// TIA Portal project "scada ile istasyon ürün ayırma factoriy io" (V16)
// Vorlageprojekt für das Buch mit Zielsystem S7-1200

(* hardware
DEVICE "S7-1200-Station_1"  S7-1200 Station
   slot 0: "Baugruppenträger_0"  Rack  V1.0
   slot 1: "PLC_1"  CPU 1214C DC/DC/DC  6ES7 214-1AG40-0XB0  V4.4
   slot 2: "AQ 2x14BIT_1"  SM 1232 AQ2  6ES7 232-4HB32-0XB0  V2.1
DEVICE "PC-System_1"  SIMATIC PC station
   slot 0: "SIMATIC PC station"  Rail  SIMATIC PC-Station  V1.0
      slot 125: "Stationmanager"  Station_Manager  V6.0.4
   slot 1: "HMI_RT_1"  WinCC RT Professional  6AV2 105-0xxxx-xxxx  16.0.0.0
   slot 2: "IE general_1"  IE General  IE_CP  V8.2.0
*)

// ===== PLC "PLC_1"  CPU 1214C DC/DC/DC =====

VAR_GLOBAL   // PLC tag table "ANALOG İNPUTLAR"
   "GÖRÜNTÜ SENSÖRÜ 1" AT %IW30 : Int;
   "GÖRÜNTÜ SENSÖRÜ 2" AT %IW32 : Int;
END_VAR

VAR_GLOBAL   // PLC tag table "OUTPUTLAR"
   "AYIRICI 1" AT %Q0.0 : Bool;
   "AYIRICI 2" AT %Q0.1 : Bool;
   "KONVEYÖR  1" AT %Q0.2 : Bool;
   "KONVEYÖR  2" AT %Q0.3 : Bool;
   "KONVEYÖR  3" AT %Q0.4 : Bool;
   "KONVEYÖR  4" AT %Q0.5 : Bool;
END_VAR

VAR_GLOBAL   // PLC tag table "İNPUTLAR"
   "SENSÖR 1" AT %I0.0 : Bool;
   "SENSÖR 2" AT %I0.1 : Bool;
   "SENSÖR 3" AT %I0.2 : Bool;
   "SENSÖR 4" AT %I0.3 : Bool;
   "AYIRICI 1 GERİ SENSÖRÜ" AT %I0.4 : Bool;
   "AYIRICI 1 İLERİ SENSÖRÜ" AT %I0.5 : Bool;
   "AYIRICI 2 GERİ SENSÖRÜ" AT %I0.6 : Bool;
   "AYIRICI 2 İLERİ SENSÖRÜ" AT %I0.7 : Bool;
END_VAR

DATA_BLOCK "DATALAR"   // DB1
{ S7_Optimized_Access := 'TRUE' }
VERSION : 0.1
   VAR
      "SİSTEM START" : Bool;
      "SİSTEM STOP" : Bool;
      "SİSTEM RESET" : Bool;
      "SİSTEM GENEL MEM" : Bool;
      "YESİL ÜRÜN SAYISI" : Int;
      "MAVİ ÜRÜN SAYISI" : Int;
      "TOPLAM ÜRÜN SAYISI" : Int;
      "AYRILACAK ÜRÜN SAYISI" : Int;
      M1 : Bool;
      M2 : Bool;
      M3 : Bool;
      M4 : Bool;
      "AYRICI DURUM BİL MEM" : Bool;
      "M3_GRT 1 MAVİ" : Bool;
      "M3_GRT 1 YESİL" : Bool;
      "M3_GRT  2 MAVİ" : Bool;
      "M3_GRT 2  YESİL" : Bool;
      TEMP_1 : Bool;
      TEMP_2 : Bool;
      TEMP_3 : Bool;
      TEMP_4 : Bool;
      TEMP_5 : Bool;
      TEMP_6 : Bool;
      TEMP_7 : Bool;
      TEMP_8 : Bool;
      TEMP_9 : Bool;
   END_VAR
BEGIN
END_DATA_BLOCK

// folder: System blocks/Program resources

DATA_BLOCK "TİME 1"   // DB2
{ S7_Optimized_Access := 'TRUE' }
AUTHOR : Simatic
FAMILY : IEC
NAME : IEC_TMR
VERSION : 1.0
// stored: InstanceOfName IEC_TIMER
"IEC_TIMER"
BEGIN
END_DATA_BLOCK

DATA_BLOCK "TİME 2"   // DB3
{ S7_Optimized_Access := 'TRUE' }
AUTHOR : Simatic
FAMILY : IEC
NAME : IEC_TMR
VERSION : 1.0
// stored: InstanceOfName IEC_TIMER
"IEC_TIMER"
BEGIN
END_DATA_BLOCK

DATA_BLOCK "tİME 3"   // DB4
{ S7_Optimized_Access := 'TRUE' }
AUTHOR : Simatic
FAMILY : IEC
NAME : IEC_TMR
VERSION : 1.0
// stored: InstanceOfName IEC_TIMER
"IEC_TIMER"
BEGIN
END_DATA_BLOCK

DATA_BLOCK "SAYICI 1"   // DB5
{ S7_Optimized_Access := 'TRUE' }
AUTHOR : Simatic
FAMILY : IEC
NAME : CNTR
VERSION : 1.0
// stored: InstanceOfName IEC_COUNTER
"IEC_COUNTER"
BEGIN
END_DATA_BLOCK

// folder: (top level)

FUNCTION "MHJ-PLC-Lab-Function-S71200" : Void   // FC9000, SCL
{ S7_Optimized_Access := 'TRUE' }
VERSION : 0.1
   VAR_TEMP
      rdTimeReturn : Int;
      outputTime : DTL;
      SyncVal : Byte;
      forVal : Int;
      forVal_2 : Int;
      Value : Byte;
   END_VAR
   VAR CONSTANT
      CompVal : Byte := 16#34;
      Value_01 : Byte := 16#11;
      Value_01_DW : DWord := 16#A165_D992;
      Value_02_DW : DWord := 16#58BE_4401;
   END_VAR
BEGIN

   #Value:=PEEK(area := 16#82,
        dbNumber := 0,
        byteOffset := 511);
   #Value := #Value + 1;

   POKE(area := 16#82,
        dbNumber := 0,
        byteOffset := 511,
        value := #Value);

   POKE(area:=16#81,
        dbNumber:=0,
        byteOffset:=1016,
        value:=#Value_01_DW);
   POKE(area := 16#81,
        dbNumber := 0,
        byteOffset := 1020,
        value := #Value_02_DW);

   POKE(area := 16#81,
        dbNumber := 0,
        byteOffset := 511,
        value := B#16#00);

   FOR #forVal := 0 TO 120 DO
       FOR #forVal_2:=0 TO 10 DO
           #rdTimeReturn:=RD_SYS_T(#outputTime);
           #rdTimeReturn := WR_SYS_T(#outputTime);
           #rdTimeReturn := RD_SYS_T(#outputTime);
           #rdTimeReturn := WR_SYS_T(#outputTime);
       END_FOR;
       #SyncVal:= PEEK(area := 16#81,
                      dbNumber := 0,
                      byteOffset := 511);
       IF #SyncVal = #CompVal THEN
          GOTO M_1;
       END_IF;
   END_FOR;
   RETURN;

   M_1:
   POKE(area := 16#81,
        dbNumber := 0,
        byteOffset := 511,
        value := B#16#0);
END_FUNCTION

ORGANIZATION_BLOCK "Main"   // OB1, LAD, ProgramCycle
TITLE = "Main Program Sweep (Cycle)"
{ S7_Optimized_Access := 'TRUE' }
VERSION : 0.1
   VAR_INPUT
      Initial_Call : Bool;   // Initial call of this OB
      Remanence : Bool;   // =True, if remanent data are available
   END_VAR
   VAR_TEMP   // added for the SCL form of the ladder/FBD networks
      _w1 : Bool;
      _w2 : Bool;
      _w3 : Bool;
   END_VAR
BEGIN

REGION Network 1: Konnektierungsbaustein für PLC-Lab
   // Im Netzwerk 1 wird der Konnektierungsbaustein für PLC-Lab aufgerufen.
   // Dieser Aufruf darf nicht entfernt werden!
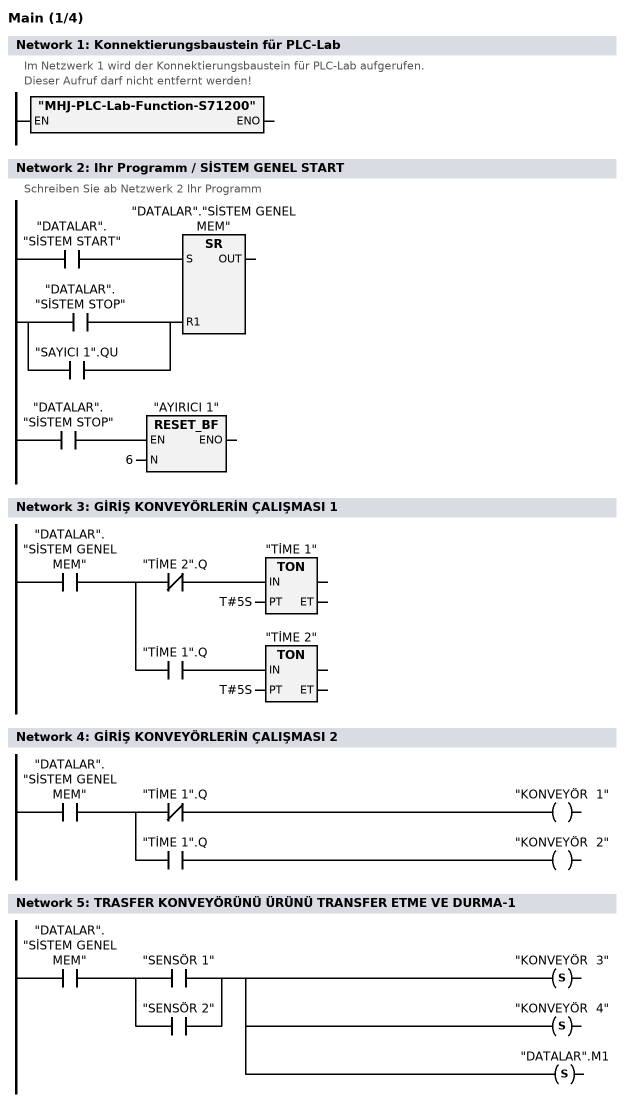
   RUNG wire#powerrail
      "MHJ-PLC-Lab-Function-S71200"()
   END_RUNG
   // the same network as SCL:
   "MHJ-PLC-Lab-Function-S71200"();
END_REGION

REGION Network 2: Ihr Programm / SİSTEM GENEL START
   // Schreiben Sie ab Netzwerk 2 Ihr Programm
   // no SCL statement known for RBitfield: written as a call
   IF "DATALAR"."SİSTEM START" THEN
       "DATALAR"."SİSTEM GENEL MEM" := TRUE;   // SR flip-flop
   END_IF;
   IF "DATALAR"."SİSTEM STOP" OR "SAYICI 1".QU THEN "DATALAR"."SİSTEM GENEL MEM" := FALSE; END_IF;
   IF "DATALAR"."SİSTEM STOP" THEN RESET_BF(operand := "AYIRICI 1", n := 6); END_IF;
END_REGION

REGION Network 3: GİRİŞ KONVEYÖRLERİN ÇALIŞMASI 1
   "TİME 1".TON(IN := "DATALAR"."SİSTEM GENEL MEM" AND NOT "TİME 2".Q, PT := T#5S);
   "TİME 2".TON(IN := "DATALAR"."SİSTEM GENEL MEM" AND "TİME 1".Q, PT := T#5S);
END_REGION

REGION Network 4: GİRİŞ KONVEYÖRLERİN ÇALIŞMASI 2
   RUNG wire#powerrail
      Contact( "DATALAR"."SİSTEM GENEL MEM" )
      wire#w1
      I_Contact( "TİME 1".Q )
      Coil( "KONVEYÖR  1" )
   END_RUNG
   RUNG wire#w1
      Contact( "TİME 1".Q )
      Coil( "KONVEYÖR  2" )
   END_RUNG
   // the same network as SCL:
   "KONVEYÖR  1" := "DATALAR"."SİSTEM GENEL MEM" AND NOT "TİME 1".Q;
   "KONVEYÖR  2" := "DATALAR"."SİSTEM GENEL MEM" AND "TİME 1".Q;
END_REGION

REGION Network 5: TRASFER KONVEYÖRÜNÜ ÜRÜNÜ TRANSFER ETME VE DURMA-1
   RUNG wire#powerrail
      Contact( "DATALAR"."SİSTEM GENEL MEM" )
      wire#w1
      Contact( "SENSÖR 1" )
      wire#w2
      S_Coil( "KONVEYÖR  3" )
   END_RUNG
   RUNG wire#w1
      Contact( "SENSÖR 2" )
   END_RUNG wire#w2
   RUNG wire#w2
      S_Coil( "KONVEYÖR  4" )
   END_RUNG
   RUNG wire#w2
      S_Coil( "DATALAR".M1 )
   END_RUNG
   // the same network as SCL:
   IF "DATALAR"."SİSTEM GENEL MEM" AND ("SENSÖR 1" OR "SENSÖR 2") THEN
       "KONVEYÖR  3" := TRUE;
       "KONVEYÖR  4" := TRUE;
       "DATALAR".M1 := TRUE;
   END_IF;
END_REGION

REGION Network 6: TRASFER KONVEYÖRÜNÜ ÜRÜNÜ TRANSFER ETME VE DURMA-2
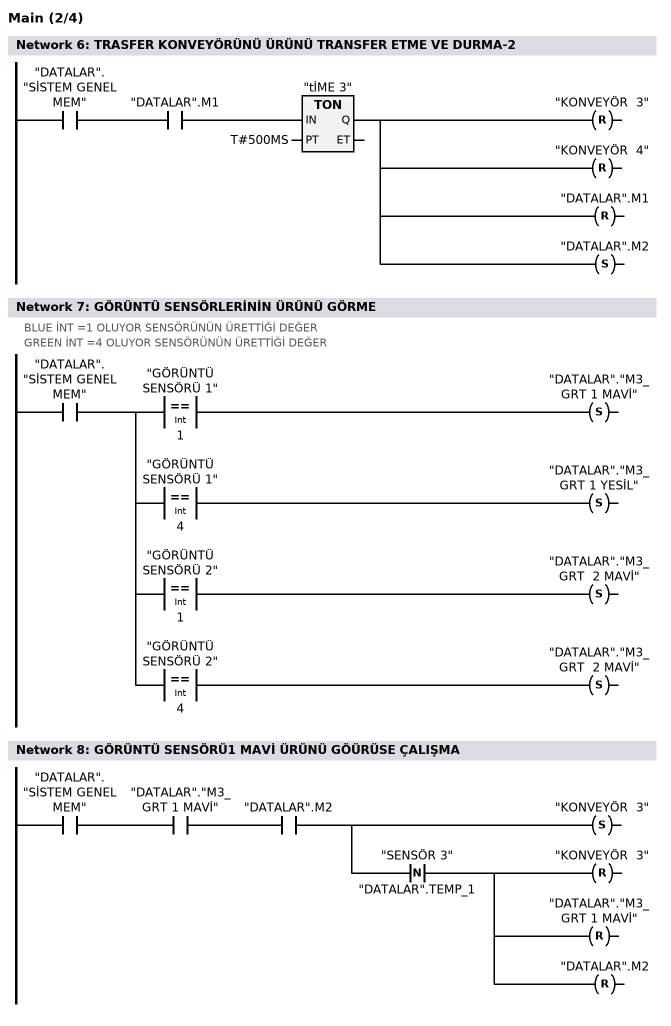
   "tİME 3".TON(IN := "DATALAR"."SİSTEM GENEL MEM" AND "DATALAR".M1, PT := T#500MS);
   IF "tİME 3".Q THEN
       "KONVEYÖR  3" := FALSE;
       "KONVEYÖR  4" := FALSE;
       "DATALAR".M1 := FALSE;
       "DATALAR".M2 := TRUE;
   END_IF;
END_REGION

REGION Network 7: GÖRÜNTÜ SENSÖRLERİNİN ÜRÜNÜ GÖRME
   // BLUE İNT =1 OLUYOR SENSÖRÜNÜN ÜRETTİĞİ DEĞER
   // GREEN İNT =4 OLUYOR SENSÖRÜNÜN ÜRETTİĞİ DEĞER
   RUNG wire#powerrail
      Contact( "DATALAR"."SİSTEM GENEL MEM" )
      wire#w1
      { S7_Templates := "SrcType := Int" } EQ_Contact(in1 := "GÖRÜNTÜ SENSÖRÜ 1", in2 := 1)
      S_Coil( "DATALAR"."M3_GRT 1 MAVİ" )
   END_RUNG
   RUNG wire#w1
      { S7_Templates := "SrcType := Int" } EQ_Contact(in1 := "GÖRÜNTÜ SENSÖRÜ 1", in2 := 4)
      S_Coil( "DATALAR"."M3_GRT 1 YESİL" )
   END_RUNG
   RUNG wire#w1
      { S7_Templates := "SrcType := Int" } EQ_Contact(in1 := "GÖRÜNTÜ SENSÖRÜ 2", in2 := 1)
      S_Coil( "DATALAR"."M3_GRT  2 MAVİ" )
   END_RUNG
   RUNG wire#w1
      { S7_Templates := "SrcType := Int" } EQ_Contact(in1 := "GÖRÜNTÜ SENSÖRÜ 2", in2 := 4)
      S_Coil( "DATALAR"."M3_GRT  2 MAVİ" )
   END_RUNG
   // the same network as SCL:
   IF "DATALAR"."SİSTEM GENEL MEM" AND ("GÖRÜNTÜ SENSÖRÜ 1" = 1) THEN
       "DATALAR"."M3_GRT 1 MAVİ" := TRUE;
   END_IF;
   IF "DATALAR"."SİSTEM GENEL MEM" AND ("GÖRÜNTÜ SENSÖRÜ 1" = 4) THEN
       "DATALAR"."M3_GRT 1 YESİL" := TRUE;
   END_IF;
   IF "DATALAR"."SİSTEM GENEL MEM" AND ("GÖRÜNTÜ SENSÖRÜ 2" = 1) THEN
       "DATALAR"."M3_GRT  2 MAVİ" := TRUE;
   END_IF;
   IF "DATALAR"."SİSTEM GENEL MEM" AND ("GÖRÜNTÜ SENSÖRÜ 2" = 4) THEN
       "DATALAR"."M3_GRT  2 MAVİ" := TRUE;
   END_IF;
END_REGION

REGION Network 8: GÖRÜNTÜ SENSÖRÜ1 MAVİ ÜRÜNÜ GÖÜRÜSE ÇALIŞMA
   RUNG wire#powerrail
      Contact( "DATALAR"."SİSTEM GENEL MEM" )
      Contact( "DATALAR"."M3_GRT 1 MAVİ" )
      Contact( "DATALAR".M2 )
      wire#w1
      S_Coil( "KONVEYÖR  3" )
   END_RUNG
   RUNG wire#w1
      N_Contact(operand := "SENSÖR 3", bit := "DATALAR".TEMP_1)
      wire#w2
      R_Coil( "KONVEYÖR  3" )
   END_RUNG
   RUNG wire#w2
      R_Coil( "DATALAR"."M3_GRT 1 MAVİ" )
   END_RUNG
   RUNG wire#w2
      R_Coil( "DATALAR".M2 )
   END_RUNG
   // the same network as SCL:
   #_w1 := "DATALAR"."SİSTEM GENEL MEM" AND "DATALAR"."M3_GRT 1 MAVİ" AND "DATALAR".M2;
   IF #_w1 THEN "KONVEYÖR  3" := TRUE; END_IF;
   #_w2 := #_w1 AND NOT "SENSÖR 3" AND "DATALAR".TEMP_1;   // falling edge of "SENSÖR 3"
   "DATALAR".TEMP_1 := "SENSÖR 3";
   IF #_w2 THEN
       "KONVEYÖR  3" := FALSE;
       "DATALAR"."M3_GRT 1 MAVİ" := FALSE;
       "DATALAR".M2 := FALSE;
   END_IF;
END_REGION

REGION Network 9: GÖRÜNTÜ SENSÖRÜ1 YEŞİL ÜRÜNÜ GÖÜRÜSE ÇALIŞMA
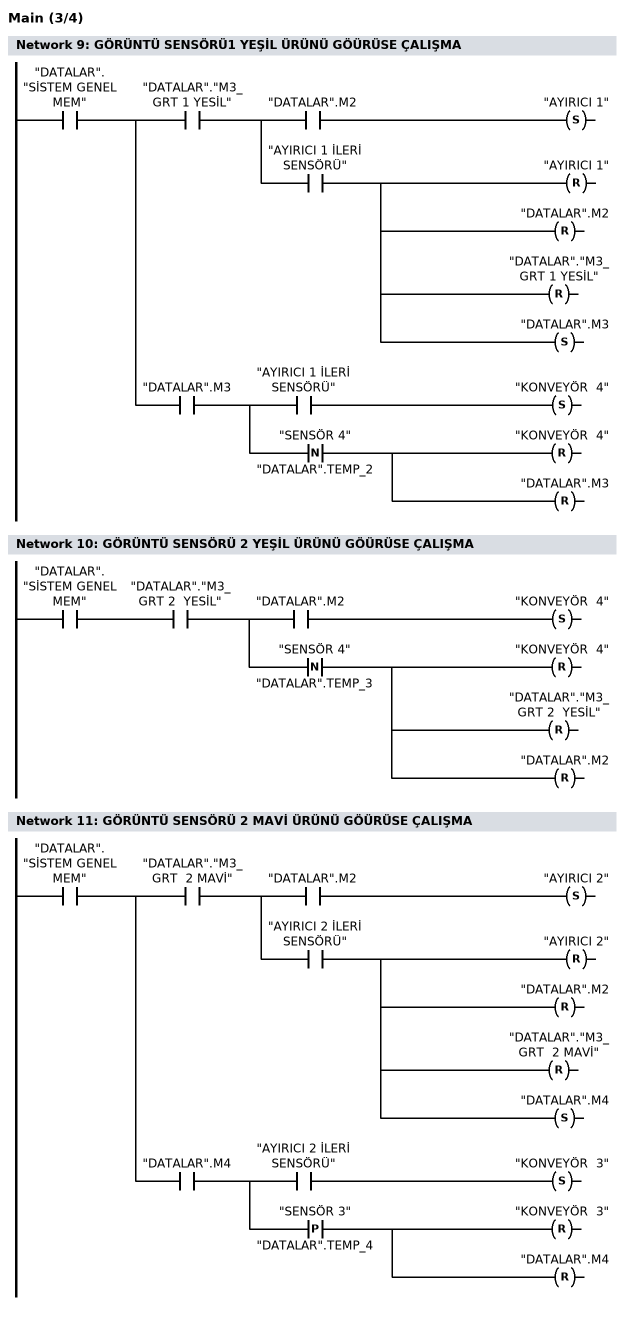
   RUNG wire#powerrail
      Contact( "DATALAR"."SİSTEM GENEL MEM" )
      wire#w1
      Contact( "DATALAR"."M3_GRT 1 YESİL" )
      wire#w2
      Contact( "DATALAR".M2 )
      S_Coil( "AYIRICI 1" )
   END_RUNG
   RUNG wire#w2
      Contact( "AYIRICI 1 İLERİ SENSÖRÜ" )
      wire#w3
      R_Coil( "AYIRICI 1" )
   END_RUNG
   RUNG wire#w3
      R_Coil( "DATALAR".M2 )
   END_RUNG
   RUNG wire#w3
      R_Coil( "DATALAR"."M3_GRT 1 YESİL" )
   END_RUNG
   RUNG wire#w3
      S_Coil( "DATALAR".M3 )
   END_RUNG
   RUNG wire#w1
      Contact( "DATALAR".M3 )
      wire#w4
      Contact( "AYIRICI 1 İLERİ SENSÖRÜ" )
      S_Coil( "KONVEYÖR  4" )
   END_RUNG
   RUNG wire#w4
      N_Contact(operand := "SENSÖR 4", bit := "DATALAR".TEMP_2)
      wire#w5
      R_Coil( "KONVEYÖR  4" )
   END_RUNG
   RUNG wire#w5
      R_Coil( "DATALAR".M3 )
   END_RUNG
   // the same network as SCL:
   #_w1 := "DATALAR"."SİSTEM GENEL MEM" AND "DATALAR"."M3_GRT 1 YESİL";
   IF #_w1 AND "DATALAR".M2 THEN "AYIRICI 1" := TRUE; END_IF;
   IF #_w1 AND "AYIRICI 1 İLERİ SENSÖRÜ" THEN
       "AYIRICI 1" := FALSE;
       "DATALAR".M2 := FALSE;
       "DATALAR"."M3_GRT 1 YESİL" := FALSE;
       "DATALAR".M3 := TRUE;
   END_IF;
   #_w2 := "DATALAR"."SİSTEM GENEL MEM" AND "DATALAR".M3;
   IF #_w2 AND "AYIRICI 1 İLERİ SENSÖRÜ" THEN "KONVEYÖR  4" := TRUE; END_IF;
   #_w3 := #_w2 AND NOT "SENSÖR 4" AND "DATALAR".TEMP_2;   // falling edge of "SENSÖR 4"
   "DATALAR".TEMP_2 := "SENSÖR 4";
   IF #_w3 THEN
       "KONVEYÖR  4" := FALSE;
       "DATALAR".M3 := FALSE;
   END_IF;
END_REGION

REGION Network 10: GÖRÜNTÜ SENSÖRÜ 2 YEŞİL ÜRÜNÜ GÖÜRÜSE ÇALIŞMA
   RUNG wire#powerrail
      Contact( "DATALAR"."SİSTEM GENEL MEM" )
      Contact( "DATALAR"."M3_GRT 2  YESİL" )
      wire#w1
      Contact( "DATALAR".M2 )
      S_Coil( "KONVEYÖR  4" )
   END_RUNG
   RUNG wire#w1
      N_Contact(operand := "SENSÖR 4", bit := "DATALAR".TEMP_3)
      wire#w2
      R_Coil( "KONVEYÖR  4" )
   END_RUNG
   RUNG wire#w2
      R_Coil( "DATALAR"."M3_GRT 2  YESİL" )
   END_RUNG
   RUNG wire#w2
      R_Coil( "DATALAR".M2 )
   END_RUNG
   // the same network as SCL:
   #_w1 := "DATALAR"."SİSTEM GENEL MEM" AND "DATALAR"."M3_GRT 2  YESİL";
   IF #_w1 AND "DATALAR".M2 THEN "KONVEYÖR  4" := TRUE; END_IF;
   #_w2 := #_w1 AND NOT "SENSÖR 4" AND "DATALAR".TEMP_3;   // falling edge of "SENSÖR 4"
   "DATALAR".TEMP_3 := "SENSÖR 4";
   IF #_w2 THEN
       "KONVEYÖR  4" := FALSE;
       "DATALAR"."M3_GRT 2  YESİL" := FALSE;
       "DATALAR".M2 := FALSE;
   END_IF;
END_REGION

REGION Network 11: GÖRÜNTÜ SENSÖRÜ 2 MAVİ ÜRÜNÜ GÖÜRÜSE ÇALIŞMA
   RUNG wire#powerrail
      Contact( "DATALAR"."SİSTEM GENEL MEM" )
      wire#w1
      Contact( "DATALAR"."M3_GRT  2 MAVİ" )
      wire#w2
      Contact( "DATALAR".M2 )
      S_Coil( "AYIRICI 2" )
   END_RUNG
   RUNG wire#w2
      Contact( "AYIRICI 2 İLERİ SENSÖRÜ" )
      wire#w3
      R_Coil( "AYIRICI 2" )
   END_RUNG
   RUNG wire#w3
      R_Coil( "DATALAR".M2 )
   END_RUNG
   RUNG wire#w3
      R_Coil( "DATALAR"."M3_GRT  2 MAVİ" )
   END_RUNG
   RUNG wire#w3
      S_Coil( "DATALAR".M4 )
   END_RUNG
   RUNG wire#w1
      Contact( "DATALAR".M4 )
      wire#w4
      Contact( "AYIRICI 2 İLERİ SENSÖRÜ" )
      S_Coil( "KONVEYÖR  3" )
   END_RUNG
   RUNG wire#w4
      P_Contact(operand := "SENSÖR 3", bit := "DATALAR".TEMP_4)
      wire#w5
      R_Coil( "KONVEYÖR  3" )
   END_RUNG
   RUNG wire#w5
      R_Coil( "DATALAR".M4 )
   END_RUNG
   // the same network as SCL:
   #_w1 := "DATALAR"."SİSTEM GENEL MEM" AND "DATALAR"."M3_GRT  2 MAVİ";
   IF #_w1 AND "DATALAR".M2 THEN "AYIRICI 2" := TRUE; END_IF;
   IF #_w1 AND "AYIRICI 2 İLERİ SENSÖRÜ" THEN
       "AYIRICI 2" := FALSE;
       "DATALAR".M2 := FALSE;
       "DATALAR"."M3_GRT  2 MAVİ" := FALSE;
       "DATALAR".M4 := TRUE;
   END_IF;
   #_w2 := "DATALAR"."SİSTEM GENEL MEM" AND "DATALAR".M4;
   IF #_w2 AND "AYIRICI 2 İLERİ SENSÖRÜ" THEN "KONVEYÖR  3" := TRUE; END_IF;
   #_w3 := #_w2 AND "SENSÖR 3" AND NOT "DATALAR".TEMP_4;   // rising edge of "SENSÖR 3"
   "DATALAR".TEMP_4 := "SENSÖR 3";
   IF #_w3 THEN
       "KONVEYÖR  3" := FALSE;
       "DATALAR".M4 := FALSE;
   END_IF;
END_REGION

REGION Network 12: AYRILAN ÜRÜNLERİ SAYMA
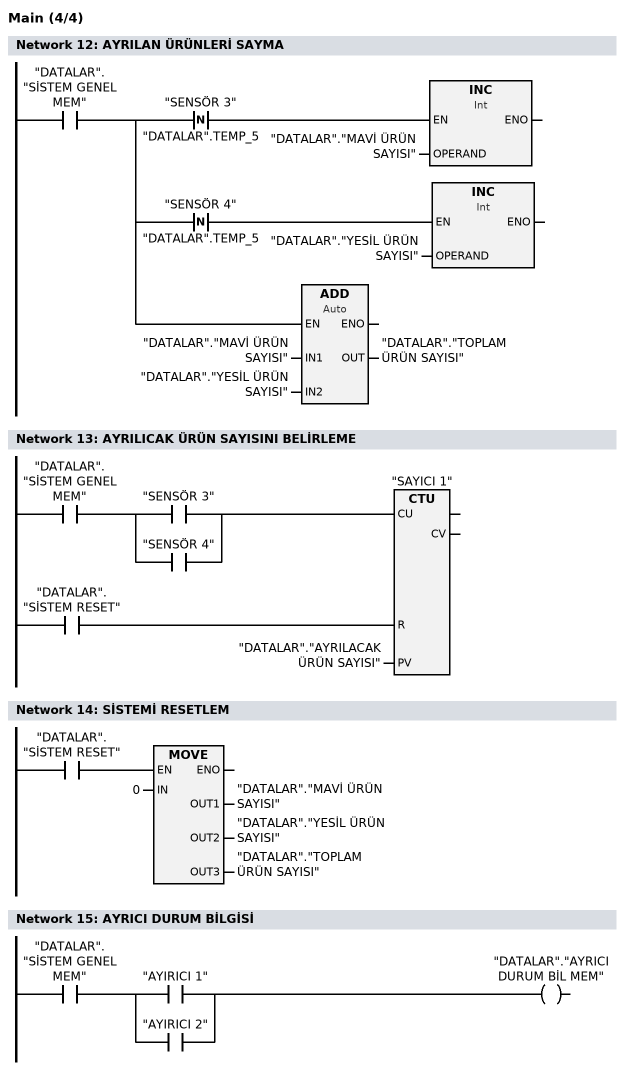
   RUNG wire#powerrail
      Contact( "DATALAR"."SİSTEM GENEL MEM" )
      wire#w1
      N_Contact(operand := "SENSÖR 3", bit := "DATALAR".TEMP_5)
      { S7_Templates := "DestType := Int" } Inc( "DATALAR"."MAVİ ÜRÜN SAYISI" )
   END_RUNG
   RUNG wire#w1
      N_Contact(operand := "SENSÖR 4", bit := "DATALAR".TEMP_5)
      { S7_Templates := "DestType := Int" } Inc( "DATALAR"."YESİL ÜRÜN SAYISI" )
   END_RUNG
   RUNG wire#w1
      Add(in1 := "DATALAR"."MAVİ ÜRÜN SAYISI", in2 := "DATALAR"."YESİL ÜRÜN SAYISI", out => "DATALAR"."TOPLAM ÜRÜN SAYISI")
   END_RUNG
   // the same network as SCL:
   #_w1 := "DATALAR"."SİSTEM GENEL MEM" AND NOT "SENSÖR 3" AND "DATALAR".TEMP_5;   // falling edge of "SENSÖR 3"
   "DATALAR".TEMP_5 := "SENSÖR 3";
   IF #_w1 THEN "DATALAR"."MAVİ ÜRÜN SAYISI" := "DATALAR"."MAVİ ÜRÜN SAYISI" + 1; END_IF;
   #_w2 := "DATALAR"."SİSTEM GENEL MEM" AND NOT "SENSÖR 4" AND "DATALAR".TEMP_5;   // falling edge of "SENSÖR 4"
   "DATALAR".TEMP_5 := "SENSÖR 4";
   IF #_w2 THEN "DATALAR"."YESİL ÜRÜN SAYISI" := "DATALAR"."YESİL ÜRÜN SAYISI" + 1; END_IF;
   IF "DATALAR"."SİSTEM GENEL MEM" THEN
       "DATALAR"."TOPLAM ÜRÜN SAYISI" := "DATALAR"."MAVİ ÜRÜN SAYISI" + "DATALAR"."YESİL ÜRÜN SAYISI";
   END_IF;
END_REGION

REGION Network 13: AYRILICAK ÜRÜN SAYISINI BELİRLEME
   "SAYICI 1".CTU(CU := "DATALAR"."SİSTEM GENEL MEM" AND ("SENSÖR 3" OR "SENSÖR 4"),
                  R := "DATALAR"."SİSTEM RESET",
                  PV := "DATALAR"."AYRILACAK ÜRÜN SAYISI");
END_REGION

REGION Network 14: SİSTEMİ RESETLEM
   RUNG wire#powerrail
      Contact( "DATALAR"."SİSTEM RESET" )
      Move(in := 0, out1 => "DATALAR"."MAVİ ÜRÜN SAYISI", out2 => "DATALAR"."YESİL ÜRÜN SAYISI", out3 => "DATALAR"."TOPLAM ÜRÜN SAYISI")
   END_RUNG
   // the same network as SCL:
   IF "DATALAR"."SİSTEM RESET" THEN
       "DATALAR"."MAVİ ÜRÜN SAYISI" := 0;
       "DATALAR"."YESİL ÜRÜN SAYISI" := 0;
       "DATALAR"."TOPLAM ÜRÜN SAYISI" := 0;
   END_IF;
END_REGION

REGION Network 15: AYRICI DURUM BİLGİSİ
   RUNG wire#powerrail
      Contact( "DATALAR"."SİSTEM GENEL MEM" )
      wire#w1
      Contact( "AYIRICI 1" )
      wire#w2
      Coil( "DATALAR"."AYRICI DURUM BİL MEM" )
   END_RUNG
   RUNG wire#w1
      Contact( "AYIRICI 2" )
   END_RUNG wire#w2
   // the same network as SCL:
   "DATALAR"."AYRICI DURUM BİL MEM" := "DATALAR"."SİSTEM GENEL MEM" AND ("AYIRICI 1" OR "AYIRICI 2");
END_REGION
END_ORGANIZATION_BLOCK

(* ===== HMI "HMI_RT_1" =====
system functions are stored by id; their names below are inferred from use
connection "HMI_Connection_1": S71200_TCP_IP, SCADA_S7_1200

HMI tags "Default tag table"
   "1" : Bool = PLC 1 AT %I0.0, 500 ms
   "DATALAR_SİSTEMSTART" : Bool = PLC DATALAR."SİSTEM START", 500 ms
   "DATALAR_SİSTEMSTOP" : Bool = PLC DATALAR."SİSTEM STOP", 500 ms
   "DATALAR_SİSTEMRESET" : Bool = PLC DATALAR."SİSTEM RESET", 500 ms
   "DATALAR_MAVİÜRÜNSAYISI" : Int = PLC DATALAR."MAVİ ÜRÜN SAYISI", 500 ms
   "DATALAR_YESİLÜRÜNSAYISI" : Int = PLC DATALAR."YESİL ÜRÜN SAYISI", 500 ms
   "DATALAR_TOPLAMÜRÜNSAYISI" : Int = PLC DATALAR."TOPLAM ÜRÜN SAYISI", 500 ms
   "DATALAR_SİSTEMGENELMEM" : Bool = PLC DATALAR."SİSTEM GENEL MEM", 500 ms
   "DATALAR_AYRILACAKÜRÜNSAYISI" : Int = PLC DATALAR."AYRILACAK ÜRÜN SAYISI", 500 ms
   "DATALAR_AYRICIDURUMBİLMEM" : Bool = PLC DATALAR."AYRICI DURUM BİL MEM", 500 ms

screen "Screen_1" 1024x768
   TextField "Text field_1" at 332,9 size 298x28; Text 'ÜRÜN AYIRMA İSTASYONU'
   IOField "I/O field_1" at 184,114 size 107x37; FormatPattern 9999
      ProcessValue <- "DATALAR_MAVİÜRÜNSAYISI"
   TextField "Text field_2" at 179,80 size 143x19; Text 'MAVİ ÜRÜN SAYISI'
   IOField "I/O field_2" at 398,111 size 107x37; FormatPattern 9999
      ProcessValue <- "DATALAR_YESİLÜRÜNSAYISI"
   TextField "Text field_3" at 382,78 size 146x19; Text 'YESİL ÜRÜN SAYISI'
   IOField "I/O field_3" at 627,110 size 107x37; FormatPattern 999
      ProcessValue <- "DATALAR_TOPLAMÜRÜNSAYISI"
   TextField "Text field_4" at 599,78 size 166x19; Text 'TOPLAM ÜRÜN SAYISI'
   Button "Button_1" at 156,179 size 161x66; TextOff 'SİSTEM START'
      on PressLeft: SetBit("DATALAR_SİSTEMSTART")
      on ReleaseLeft: ResetBit("DATALAR_SİSTEMSTART")
      Appearance <- "DATALAR_SİSTEMSTART"
   Button "Button_2" at 382,179 size 157x66; TextOff 'SİSTEM STOP'
      on PressLeft: SetBit("DATALAR_SİSTEMSTOP")
      on ReleaseLeft: ResetBit("DATALAR_SİSTEMSTOP")
      Appearance <- "DATALAR_SİSTEMSTOP"
   Button "Button_3" at 612,179 size 157x66; TextOff 'SİSTEM RESET'
      on PressLeft: SetBit("DATALAR_SİSTEMRESET")
      on ReleaseLeft: ResetBit("DATALAR_SİSTEMRESET")
      Appearance <- "DATALAR_SİSTEMRESET"
   TextField "Text field_5" at 386,300 size 170x23; Text 'SİSTEM ÇALIŞIYOR'
      Visibility <- "DATALAR_SİSTEMGENELMEM"
   TextField "Text field_6" at 386,300 size 163x23; Text 'SİSTEM DURUYOR'
      Visibility <- "DATALAR_SİSTEMGENELMEM"
   IOField "I/O field_4" at 407,699 size 111x39; FormatPattern 999
      ProcessValue <- "DATALAR_AYRILACAKÜRÜNSAYISI"
   TextField "Text field_7" at 391,668 size 185x19; Text 'AYRILICAK ÜRÜN SAYISI'
   GraphicView "Graphic view_1" at 357,363 size 250x250; Picture "Graphic_20"
      Visibility <- "DATALAR_AYRICIDURUMBİLMEM"
   GraphicView "Graphic view_2" at 357,363 size 250x250; Picture "Graphic_21"
      Visibility <- "DATALAR_AYRICIDURUMBİLMEM"
*)